{region '#Template'}
	{attribute 'Version' := '6.0.0.0'}
	{attribute 'Tags' := '"LCID": "1031", "Text": "AC, Aggregate, Ventilator"'}
	{attribute 'Tags' := '"LCID": "1033", "Text": "AC, Aggregate, Fan"'}
	{attribute 'Using' := '"Type": "Template", "URI": "Priority"'}		 
	{attribute 'Using' := '"Type": "Template", "URI": "EC_ID"'}
	{attribute 'Using' := '"Type": "Template", "URI": "BA2_Param"'}
	{attribute 'Description' := '"LCID": "1031", "Text": "Ventilator modulierend mit Regler erweitert"'}
	{attribute 'Description' := '"LCID": "1033", "Text": "Fan modulating with controller extended"'}
{endregion}		 
FUNCTION_BLOCK FB_BA_AC_FanCtl EXTENDS FB_BA_MotCtl
VAR_INPUT
	bDamperOpen				: BOOL;
END_VAR
VAR_IN_OUT
	stAggregate				: ST_BA_Aggregate;	
END_VAR
VAR_INPUT CONSTANT
	ThOvrld					: FB_BA_BI_Raw;							
	MntnSwi					: FB_BA_BI_Raw;
	Aggregate				: FB_BA_Aggregate;																											 								
END_VAR
VAR
	PrioSwiDamper			: FB_BA_PrioSwi_UDI04;
END_VAR
VAR // added by the converter: edge detectors and wires of the graphical bodies
    _s1 : ST_BA_Mdlt;
END_VAR

Aggregate(stAggregate := stAggregate); // FB_BA_Aggregate
ThOvrld(); // FB_BA_BI_Raw
MntnSwi(); // FB_BA_BI_Raw
PrioSwiDamper(
    bEn01 := NOT bDamperOpen,
    nVal01 := E_BA_Mdlt.eOff,
    bEn03 := Aggregate.arrPriorities[Priority.nCritical],
    nVal03 := MAX(1,Aggregate.nValue)); // FB_BA_PrioSwi_UDI04
// compose _s1 : ST_BA_Mdlt
_s1.bEnSfty := Aggregate.arrPriorities[Priority.nLifeSafety];
_s1.eValSfty := MAX(1,Aggregate.nValue);
_s1.bEnCrit := PrioSwiDamper.bQ;
_s1.eValCrit := PrioSwiDamper.nVal;
_s1.bEnPgm := Aggregate.arrPriorities[Priority.nProgram];
_s1.eValPgm := MAX(1,Aggregate.nValue);
SUPER^(stCmd := _s1); // FB_BA_MotCtl

METHOD FB_init : BOOL
VAR_INPUT
	bInitRetains : BOOL; // if TRUE, the retain variables are initialized (warm start / cold start)
	bInCopyCode : BOOL;  // if TRUE, the instance afterwards gets moved into the copy code (online change)
END_VAR
ThOvrld.iParent						:= THIS^;
ThOvrld.iLabel						:= LblFun_Fault;  
ThOvrld.ePolarity					:= E_BA_Polarity.eReverse;
ThOvrld.sActiveText 				:= txtEvent_Triggered;
ThOvrld.sInactiveText 				:= txtEvent_Normal;
ThOvrld.nEventClassID				:= EC_ID.NC30;
ThOvrld.stTimeDelay.nToNormal		:= BA2_Param.nDefTimeDelay_ToNormal;
ThOvrld.stTimeDelay.nToAbnormal		:= BA2_Param.nDefTimeDelay_ToAbnormal;
ThOvrld.bAlarmValue					:= TRUE;
ThOvrld.aEventTransitionText[1]		:= txtEvent_Triggered;
ThOvrld.aEventTransitionText[2]		:= txtEvent_Error;
ThOvrld.aEventTransitionText[3]		:= txtEvent_Normal;
ThOvrld.bEventDetectionEnable		:= TRUE;
ThOvrld.eEnPlantLock				:= E_BA_LockPriority.eLocalMedium;	

MntnSwi.iParent						:= THIS^;
MntnSwi.iLabel						:= LblFun_MaintenanceMessage;  
MntnSwi.ePolarity					:= E_BA_Polarity.eReverse;
MntnSwi.sActiveText 				:= txtEvent_Maintenace;
MntnSwi.sInactiveText 				:= txtEvent_Normal;
MntnSwi.nEventClassID				:= EC_ID.NC50;
MntnSwi.stTimeDelay.nToNormal		:= BA2_Param.nDefTimeDelay_ToNormal;
MntnSwi.stTimeDelay.nToAbnormal		:= BA2_Param.nDefTimeDelay_ToAbnormal;
MntnSwi.bAlarmValue					:= TRUE;
MntnSwi.aEventTransitionText[1]		:= txtEvent_Disturb;
MntnSwi.aEventTransitionText[2]		:= txtEvent_None;
MntnSwi.aEventTransitionText[3]		:= txtEvent_Normal;
MntnSwi.bEventDetectionEnable		:= TRUE;
MntnSwi.eEnPlantLock				:= E_BA_LockPriority.eLocalMedium;
END_METHOD

END_FUNCTION_BLOCK

(* stored: Version 1.1.0.1, ProductVersion 3.1.4024.12
   POU FB_BA_AC_FanCtl: Id {ad30cb11-8207-4f17-9a40-e0f9c7e5e400}, SpecialFunc None
   Method FB_init: Id {d1ca4a82-2513-4851-beb5-e9567cd021fe} *)
